(* IEC 61131-3 sources: cc_kush_rewrite/Dumper/FC, 3 files *)

(* ---- FC_Dumper_EmergencyStop.st ---- *)
FUNCTION FC_Dumper_EmergencyStop  : BOOL
VAR_INPUT
	Dumper : ST_Dumper;
END_VAR
VAR
	j : INT := 0;
END_VAR
// Остановка моторов конвейера (унаследовано от ST_ConveyorBasic)
FOR j := 1 TO 2 DO
	Dumper.MotorConveyor[j].qxKM_Power := FALSE;
	Dumper.MotorConveyor[j].VFD.qxStart := FALSE;
	Dumper.MotorConveyor[j].VFD.Frequency.rTargetFrequency := 0.0;
	Dumper.MotorConveyor[j].VFD.qrOutFrequency := 0.0;
END_FOR

// Остановка моторов поворота
FOR j := 1 TO 2 DO
	Dumper.MotorRotation[j].qxKM_Power := FALSE;
	Dumper.MotorRotation[j].VFD.qxStart := FALSE;
	Dumper.MotorRotation[j].VFD.Frequency.rTargetFrequency := 0.0;
	Dumper.MotorRotation[j].VFD.qrOutFrequency := 0.0;
	Dumper.MotorRotation[j].qxVFDReverseStart := FALSE;
END_FOR

END_FUNCTION

(* ---- FC_Dumper_GetErrorCommon.st ---- *)
FUNCTION FC_Dumper_GetErrorCommon : BOOL
VAR_INPUT
	Dumper : REFERENCE TO ST_Dumper;
END_VAR
VAR
END_VAR
FC_Dumper_GetErrorCommon :=
	FC_Dumper_GetErrorSensors(Dumper := Dumper)
	OR FC_Conveyor_GetErrorMotor(motor := Dumper.MotorConveyor[1])
	OR FC_Conveyor_GetErrorMotor(motor := Dumper.MotorConveyor[2])
	OR FC_Conveyor_GetErrorMotor(motor := Dumper.MotorRotation[1])
	OR FC_Conveyor_GetErrorMotor(motor := Dumper.MotorRotation[2]);

END_FUNCTION

(* ---- FC_Dumper_GetErrorSensors.st ---- *)
FUNCTION FC_Dumper_GetErrorSensors : BOOL
VAR_INPUT
	Dumper : REFERENCE TO ST_Dumper;
END_VAR
VAR
END_VAR
FC_Dumper_GetErrorSensors := (
	// Контроль схода ленты - тревога
	FC_Sensor_CheckZQAlarm(fbZQAlarm := Dumper.fbZQAlarm)
	// Кабель-тросовый выключатель
	OR FC_Sensor_CheckHQ(fbHQ_IsOk := Dumper.fbHQ_IsOk)
	// Контроль ограждения барабана
	OR FC_Sensor_CheckSQ(fbSQ_IsOk := Dumper.fbSQ_IsOk)
	// Контроль заштыбовки
	OR FC_Sensor_CheckGS(fbGS := Dumper.fbGS1)
	// Контроль продольного разрыва ленты
	OR FC_Sensor_CheckYS(fbYS := Dumper.fbYS1)
);

END_FUNCTION
